// SIMATIC S7-200 project (STEP 7-Micro/WIN), CPU 222 REL 01.22

ORGANIZATION_BLOCK PRINCIPAL:OB1
TITLE=COMENTARIOS DEL PROGRAMA
BEGIN
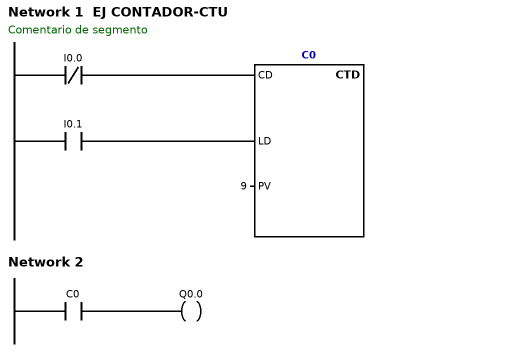
Network 1 // EJ CONTADOR-CTU

// Comentario de segmento
LDN    I0.0
LD     I0.1
CTD    C0, 9
Network 2
LD     C0
=      Q0.0
END_ORGANIZATION_BLOCK
